(* CODESYS project log-lib-all.project

Project tree, tasks and I/O mapping:
  CODESYS_Control_Win_V3 : CODESYS Control Win V3, 3S - Smart Software Solutions GmbH, order no. 305021, version 3.5.8.40
    application Application
      task MainTask (cyclic, interval t#10ms, priority 1) calls MAIN
      program MAIN [ST]
*)

// CODESYS_Control_Win_V3/Application/MAIN
PROGRAM MAIN
VAR
END_VAR

;

END_PROGRAM
